(* IEC 61131-3 sources: dynamics/src/Signals, 5 files *)

(* ---- IOutputSignal.st ---- *)
NAMESPACE Simatic.Ax.Dynamics
    /// Extends `ISignal, IOutputProvider`
    INTERFACE IOutputSignal EXTENDS ISignal, IOutputProvider
    END_INTERFACE
END_NAMESPACE

(* ---- ISignal.st ---- *)
NAMESPACE Simatic.Ax.Dynamics
    /// `Next()`
    INTERFACE ISignal
        /// Get next output
        METHOD Next : LREAL END_METHOD
    END_INTERFACE
END_NAMESPACE

(* ---- ConstantSignal.st ---- *)
NAMESPACE Simatic.Ax.Dynamics
    /// Constantly provides `output`
    CLASS ConstantSignal IMPLEMENTS IOutputSignal

        VAR PUBLIC
            /// The output value
            output : LREAL;
        END_VAR

        METHOD PUBLIC GetOutput : LREAL
            GetOutput := output;
        END_METHOD

        /// Set the output value
        METHOD PUBLIC SetOutput : LREAL
            VAR_INPUT
                newOutput : LREAL;
            END_VAR
            output := newOutput;
            SetOutput := output;
        END_METHOD

        METHOD PUBLIC Next : LREAL
            Next := THIS.GetOutput();
        END_METHOD

    END_CLASS
END_NAMESPACE

(* ---- ExplicitSignal.st ---- *)
NAMESPACE Simatic.Ax.Dynamics
    /// Signal defined by a function of the cycle number
    CLASS ABSTRACT ExplicitSignal IMPLEMENTS IOutputSignal

        VAR PRIVATE
            _cycle : UINT;
        END_VAR

        /// Reset the cycle number to zero
        METHOD PUBLIC Reset
            _cycle := UINT#0;
        END_METHOD

        /// Maps the cycle number to the output
        METHOD PROTECTED ABSTRACT _GetOutput : LREAL
            VAR_INPUT
                /// The cycle number
                cycle : UINT;
            END_VAR
        END_METHOD

        METHOD PUBLIC FINAL GetOutput : LREAL
            GetOutput := THIS._GetOutput(_cycle);
        END_METHOD

        METHOD PUBLIC FINAL Next : LREAL
            _cycle := _cycle + UINT#1;
            Next := THIS.GetOutput();
        END_METHOD

    END_CLASS
END_NAMESPACE

(* ---- RampSignal.st ---- *)
NAMESPACE Simatic.Ax.Dynamics
    /// A ramp with constant slope as given by `slope`
    /// `elapsedTimeProvider` must be set!
    CLASS RampSignal IMPLEMENTS IOutputSignal

        VAR PUBLIC
            /// The `IElapsedSecondsProvider` to use
            elapsedTimeProvider : IElapsedSecondsProvider;
            /// The slope of the ramp, being its derivative
            slope : LREAL;
        END_VAR
        VAR PRIVATE
            _output : LREAL;
        END_VAR

        METHOD PUBLIC GetOutput : LREAL
            GetOutput := _output;
        END_METHOD
        /// Set current output. Ramp will continue from there.
        METHOD PUBLIC SetOutput : LREAL
            VAR_INPUT
                newOutput : LREAL;
            END_VAR
            _output := newOutput;
            SetOutput := _output;
        END_METHOD

        /// Get the integration time T_I viewing the ramp signal as the integral over a constant signal.
        /// T_I = 1 / slope
        METHOD PUBLIC  GetTISeconds : LREAL
            GetTISeconds := 1 / slope;
        END_METHOD

        /// Set the integration time T_I viewing the ramp signal as the integral over a constant signal.
        /// T_I = 1 / slope
        METHOD PUBLIC SetTISeconds
            VAR_INPUT
                newTISeconds : LREAL;
            END_VAR
            slope := 1 / newTISeconds;
        END_METHOD

        METHOD PUBLIC Next : LREAL
            _output := _output + elapsedTimeProvider.GetElapsedSeconds() * slope;
            Next := _output;
        END_METHOD

    END_CLASS
END_NAMESPACE
